# EPICS substitutions: cpswAsynPortDriverApp/Db/testAsynPortDriver.substitutions
file testAsynPortDriver.template
{
    pattern { NAME , driver}
    { Temperature , AxiXadc}
    { VccInt , AxiXadc}
    { VccAux , AxiXadc}
    { Vin , AxiXadc}
    { VrefP , AxiXadc}
    { VrefN , AxiXadc}
    { VccBram , AxiXadc}
    { SupplyOffsetA , AxiXadc}
    { AdcOffsetA , AxiXadc}
    { AdcGainA , AxiXadc}
    { VccpInt , AxiXadc}
    { VccpAux , AxiXadc}
    { VccpDdr , AxiXadc}
    { VinAux00 , AxiXadc}
    { VinAux01 , AxiXadc}
    { VinAux02 , AxiXadc}
    { VinAux03 , AxiXadc}
    { VinAux04 , AxiXadc}
    { VinAux05 , AxiXadc}
    { VinAux06 , AxiXadc}
    { VinAux07 , AxiXadc}
    { VinAux08 , AxiXadc}
    { VinAux09 , AxiXadc}
    { VinAux10 , AxiXadc}
    { VinAux11 , AxiXadc}
    { VinAux12 , AxiXadc}
    { VinAux13 , AxiXadc}
    { VinAux14 , AxiXadc}
    { VinAux15 , AxiXadc}
    { TemperatureMax  , AxiXadc}
    { VccIntMax , AxiXadc}
    { VccAuxMax , AxiXadc}
    { VccBramMax , AxiXadc}
    { TemperatureMin , AxiXadc}
    { VccIntMin , AxiXadc}
    { VccAuxMin , AxiXadc}
    { VccBramMin , AxiXadc}
    { VccpIntMax , AxiXadc}
    { VccpAuxMax , AxiXadc}
    { VccpDdrMax , AxiXadc}
    { VccpIntMin , AxiXadc}
    { VccpAuxMin , AxiXadc}
    { VccpDdrMin , AxiXadc}
    { Flag , AxiXadc}
    { VccpIntMax , AxiXadc}

    {FpgaVersion, AxiVersion}
    {ScratchPad, AxiVersion}
    {DeviceDnaHigh, AxiVersion}
    {DeviceDnaLow, AxiVersion}
    {FdSerialHigh, AxiVersion}
    {FdSerialLow, AxiVersion}
    {MasterReset, AxiVersion}
    {FpgaReload, AxiVersion}
    {FpgaReloadAddress, AxiVersion}
    {Counter, AxiVersion}
    {FpgaReloadHalt, AxiVersion}
    {UserConstants, AxiVersion}
}

file testAsynPortDriverWaveform.template
{
  pattern {NAME, driver}
  {BuildStamp, AxiVersion}
}
